{attribute 'qualified_only'}
{attribute 'strict'}
TYPE ERecoveryState :
(
	none := 0,
	requested := 1,
	awaiting := 2,
	running := 3,
	completed := 4,
	failed := 5
);
END_TYPE

(* stored: Version 1.1.0.1
   DUT ERecoveryState: Id {f96c2e92-0dce-481f-9f14-e6395bfdbf93} *)
